{attribute addProperty BoxType "EL6080-0000-0018"}
{attribute addProperty Id "ControlAT %Q*UINT162"}
{attribute addProperty CRC "1934178468"}
{attribute addProperty SizeInBites "16"}
{attribute addProperty SizeInBytes "2"}
TYPE Control_734938A4 :
STRUCT
	{attribute addProperty Name "Control"}
	Control AT %Q* : UINT;
END_STRUCT
END_TYPE

(* stored: Version 1.2.0.0, ProductVersion 3.1.4024.9
   DUT Control_734938A4: Id {76accf8d-c14d-4889-ac97-b98af9dea65c} *)
